TYPE T_TcpRcv : POINTER TO FB_RcvDataBuffer; END_TYPE

(* stored: Version 1.1.0.1, ProductVersion 3.1.4019.2
   DUT T_TcpRcv: Id {f9631d0d-83eb-423f-a67d-381d311ac7ed} *)
